FUNCTION_BLOCK Crane_MoveBase EXTENDS ControlPrimitiveBase
VAR_INPUT
END_VAR
VAR_OUTPUT
END_VAR
VAR
	m_ptrCrane: POINTER TO Crane;
	
	m_initDirection: BOOL; //TRUE: Clockwise, FALSE: Counterclockwise
	m_step: INT := 0;
	
	m_targettimer: TON;
	m_targetTimeout: TIME;
	

END_VAR

SUPER^();

METHOD Abort : BOOL
VAR_INPUT
END_VAR
m_ptrCrane^.METH_CarrierStop();
Abort := TRUE;
END_METHOD

METHOD AtTarget : BOOL
VAR_INPUT
END_VAR
END_METHOD

(* Execution logic of this Control Primitive. *)
METHOD PROTECTED  ExecuteInternal : BOOL
VAR_INPUT
	i_params: ParameterSet;
END_VAR
CASE m_step OF 
	0: 
		m_targettimer(IN := TRUE, PT := m_targetTimeout);
		IF AtTarget() THEN
			m_step := 2;
			m_targettimer(IN:= FALSE);
		ELSIF m_targettimer.Q THEN
			m_step := 1;
			m_targettimer(IN:= FALSE);
			m_initDirection := NOT m_initDirection;
		END_IF
		
		IF m_initDirection THEN
			m_ptrCrane^.METH_CarrierTurnClockwise();
		ELSIF NOT m_initDirection THEN
			m_ptrCrane^.METH_CarrierTurnCounterclockwise(); 
		END_IF
		
	1:
		IF AtTarget() THEN
			m_step := 2;
			m_initDirection := NOT m_initDirection;
		END_IF
		IF m_initDirection THEN
			m_ptrCrane^.METH_CarrierTurnClockwise();
		ELSIF NOT m_initDirection THEN
			m_ptrCrane^.METH_CarrierTurnCounterclockwise(); 
		END_IF
		
	2:
		m_ptrCrane^.METH_CarrierStop();
		ExecuteInternal := TRUE;
		m_step := 0;
	
END_CASE
END_METHOD

END_FUNCTION_BLOCK

(* stored: Version 1.1.0.1, ProductVersion 3.1.4024.12
   POU Crane_MoveBase: Id {69afaaf4-1d33-46e7-a69f-26343eec90e5}, SpecialFunc None
   Method Abort: Id {c8b85507-64d1-44df-ac6c-67cdb85514fd}
   Method AtTarget: Id {bf100731-5b7e-43b6-bc2f-99a9df7998b0}
   Method ExecuteInternal: Id {b95028b3-dd62-4275-adc9-87152396b9da} *)
